ABB RAPID module: tester_left.mod

MODULE tester_left
LOCAL CONST string YuMi_App_Program_Version:="1.0.1"; !Do not edit or remove this line!
LOCAL VAR robtarget s7 := [[393.368,259.451,142.731],[0.318012,-0.0912919,-0.762608,-0.555845],[-2,0,1,110],[-133.932,9E+09,9E+09,9E+09,9E+09,9E+09]];
LOCAL VAR robtarget s6 := [[-205.693,265.616,364.442],[0.26066,-0.490508,0.831316,0.0192825],[-1,-3,-3,1110],[154.417,9E+09,9E+09,9E+09,9E+09,9E+09]];
LOCAL VAR robtarget s5 := [[435.849,10.8797,372.099],[0.00792561,-0.0303329,0.92848,-0.370055],[0,3,-2,100],[6.63066,9E+09,9E+09,9E+09,9E+09,9E+09]];
LOCAL VAR robtarget s4 := [[452.446,79.9861,993.753],[0.364119,0.432144,-0.215225,0.796459],[1,-1,2,1110],[89.0425,9E+09,9E+09,9E+09,9E+09,9E+09]];
LOCAL VAR robtarget s3 := [[4.02887,190.165,514.032],[0.470931,0.100617,0.868393,0.118296],[1,-1,0,100],[5.24412,9E+09,9E+09,9E+09,9E+09,9E+09]];
LOCAL VAR robtarget s2 := [[417.707,138.41,801.923],[0.956228,0.216927,0.165802,-0.105262],[-1,0,-2,1110],[-7.30886,9E+09,9E+09,9E+09,9E+09,9E+09]];
LOCAL VAR robtarget s1 := [[474.843,467.441,660.69],[0.30573,-0.730776,-0.529535,0.30346],[1,0,-1,100],[-36.2108,9E+09,9E+09,9E+09,9E+09,9E+09]];
PROC main()
MoveSync s1;
MoveSync s2;
MoveSync s3;
MoveSync s4;
MoveSync s5;
MoveSync s6;
MoveSync s7;
ENDPROC
ENDMODULE
